# B&R Automation Studio project CleanChemi_SiteManagementSystem (part 12)

#### Status.st
```iecst
ACTION Modbus_Status_action:

	ModbusTcpMaster_HR[IdxSkids_HR]();

	//Reset Modbus buffer on connection timeout
	IF ModbusTcpMaster_HR[IdxSkids_HR].status = 50211 THEN
		brsmemset(ADR(gModbus_LR[IdxSkids_HR]),0,SIZEOF(gModbus_LR[IdxSkids_HR]));
	END_IF;

	// --------------------------------------------------------------------
	// Reset last error information
	// --------------------------------------------------------------------
	IF(reset_error) THEN
		brsmemset(ADR(ModbusTcpMaster_HR[IdxSkids_HR].last_error), 0, 2);
		reset_error := 0;
	END_IF

	// --------------------------------------------------------------------
	// Final Variable Mapping AND Data Conversion - READ
	// --------------------------------------------------------------------

	// AS Block 1 - 6000 DOSING INT
	gSkid_HR[IdxSkids_HR].Pmax_General_Variables.UNIT_ID := gModbus_HR[IdxSkids_HR].Modbus_PeroxyMAX.Block1_Int[0];
	gSkid_HR[IdxSkids_HR].Pmax_General_Variables.USER_ID := gModbus_HR[IdxSkids_HR].Modbus_PeroxyMAX.Block1_Int[2];
	gSkid_HR[IdxSkids_HR].Pmax_General_Variables.USER_ACCESS := gModbus_HR[IdxSkids_HR].Modbus_PeroxyMAX.Block1_Int[4];
	gSkid_HR[IdxSkids_HR].Pmax_General_Variables.PMAX_HOA := gModbus_HR[IdxSkids_HR].Modbus_PeroxyMAX.Block1_Int[6];
	gSkid_HR[IdxSkids_HR].Pmax_General_Variables.PMAX_STATUS := gModbus_HR[IdxSkids_HR].Modbus_PeroxyMAX.Block1_Int[8];
	gSkid_HR[IdxSkids_HR].Pmax_General_Variables.SCREEN_LOCK := INT_TO_BOOL(gModbus_HR[IdxSkids_HR].Modbus_PeroxyMAX.Block1_Int[10]);
	gSkid_HR[IdxSkids_HR].Pmax_General_Variables.HEARTBEAT := gModbus_HR[IdxSkids_HR].Modbus_PeroxyMAX.Block1_Int[12];

	gSkid_HR[IdxSkids_HR].Pmax_Pump_101.P101_XS := gModbus_HR[IdxSkids_HR].Modbus_PeroxyMAX.Block1_Int[20];
	gSkid_HR[IdxSkids_HR].Sensor_Variables.XV101 := gModbus_HR[IdxSkids_HR].Modbus_PeroxyMAX.Block1_Int[22];
	gSkid_HR[IdxSkids_HR].Sensor_Variables.XV101_ENABLE := gModbus_HR[IdxSkids_HR].Modbus_PeroxyMAX.Block1_Int[24];
	gSkid_HR[IdxSkids_HR].Pmax_Pump_101.P101_AUTOCAL := gModbus_HR[IdxSkids_HR].Modbus_PeroxyMAX.Block1_Int[26];

	gSkid_HR[IdxSkids_HR].Pmax_Pump_102.P102_XS := gModbus_HR[IdxSkids_HR].Modbus_PeroxyMAX.Block1_Int[32];
	gSkid_HR[IdxSkids_HR].Pmax_Pump_102.P102_WARN := gModbus_HR[IdxSkids_HR].Modbus_PeroxyMAX.Block1_Int[34];
	gSkid_HR[IdxSkids_HR].Pmax_Pump_102.P102_ALARM := gModbus_HR[IdxSkids_HR].Modbus_PeroxyMAX.Block1_Int[36];
	gSkid_HR[IdxSkids_HR].Sensor_Variables.XV102 := gModbus_HR[IdxSkids_HR].Modbus_PeroxyMAX.Block1_Int[38];
	gSkid_HR[IdxSkids_HR].Pmax_Pump_102.P102_AUTOCAL := gModbus_HR[IdxSkids_HR].Modbus_PeroxyMAX.Block1_Int[40];

	gSkid_HR[IdxSkids_HR].Pmax_Pump_103.P103_XS := gModbus_HR[IdxSkids_HR].Modbus_PeroxyMAX.Block1_Int[48];
	gSkid_HR[IdxSkids_HR].Pmax_Pump_103.P103_WARN := gModbus_HR[IdxSkids_HR].Modbus_PeroxyMAX.Block1_Int[50];
	gSkid_HR[IdxSkids_HR].Pmax_Pump_103.P103_ALARM := gModbus_HR[IdxSkids_HR].Modbus_PeroxyMAX.Block1_Int[52];
	gSkid_HR[IdxSkids_HR].Sensor_Variables.XV103 := gModbus_HR[IdxSkids_HR].Modbus_PeroxyMAX.Block1_Int[54];
	gSkid_HR[IdxSkids_HR].Pmax_Pump_103.P103_AUTOCAL := gModbus_HR[IdxSkids_HR].Modbus_PeroxyMAX.Block1_Int[56];

	gSkid_HR[IdxSkids_HR].Pmax_Pump_104.P104_XS := gModbus_HR[IdxSkids_HR].Modbus_PeroxyMAX.Block1_Int[64];
	gSkid_HR[IdxSkids_HR].Pmax_Pump_104.P104_WARN := gModbus_HR[IdxSkids_HR].Modbus_PeroxyMAX.Block1_Int[66];
	gSkid_HR[IdxSkids_HR].Pmax_Pump_104.P104_ALARM := gModbus_HR[IdxSkids_HR].Modbus_PeroxyMAX.Block1_Int[68];
	gSkid_HR[IdxSkids_HR].Sensor_Variables.XV104 := gModbus_HR[IdxSkids_HR].Modbus_PeroxyMAX.Block1_Int[70];
	gSkid_HR[IdxSkids_HR].Pmax_Pump_104.P104_AUTOCAL := gModbus_HR[IdxSkids_HR].Modbus_PeroxyMAX.Block1_Int[72];
	gSkid_HR[IdxSkids_HR].Pmax_Pump_104.P104_AUTOCAL_PV := gModbus_HR[IdxSkids_HR].Modbus_PeroxyMAX.Block1_Int[74];

	// AS Block 2 - 6000 DOSING INT - SPARE
	//:= gModbus_HR[IdxSkids_HR].Modbus_PeroxyMAX.Block2_Int[0];

	// AS Block 3 - 6000 DOSING REAL
	gSkid_HR[IdxSkids_HR].ConversionRatios.EFF_1:= IDEC_REAL_Conv(gModbus_HR[IdxSkids_HR].Modbus_PeroxyMAX.Block3_Real[0]);
	gSkid_HR[IdxSkids_HR].ConversionRatios.EFF_2:= IDEC_REAL_Conv(gModbus_HR[IdxSkids_HR].Modbus_PeroxyMAX.Block3_Real[1]);
	gSkid_HR[IdxSkids_HR].ConversionRatios.NAOH_TO_H2O2:= IDEC_REAL_Conv(gModbus_HR[IdxSkids_HR].Modbus_PeroxyMAX.Block3_Real[2]);
	gSkid_HR[IdxSkids_HR].ConversionRatios.TRI_TO_H2O2:= IDEC_REAL_Conv(gModbus_HR[IdxSkids_HR].Modbus_PeroxyMAX.Block3_Real[3]);
	gSkid_HR[IdxSkids_HR].ConversionRatios.NAOH_TO_TRI:= IDEC_REAL_Conv(gModbus_HR[IdxSkids_HR].Modbus_PeroxyMAX.Block3_Real[4]);

	gSkid_HR[IdxSkids_HR].Pmax_General_Variables.PMAX_CONC:= IDEC_REAL_Conv(gModbus_HR[IdxSkids_HR].Modbus_PeroxyMAX.Block3_Real[8]);
	gSkid_HR[IdxSkids_HR].Pmax_General_Variables.PMAX_RATE:= IDEC_REAL_Conv(gModbus_HR[IdxSkids_HR].Modbus_PeroxyMAX.Block3_Real[9]);
	gSkid_HR[IdxSkids_HR].Pmax_General_Variables.PMAX_PV:= IDEC_REAL_Conv(gModbus_HR[IdxSkids_HR].Modbus_PeroxyMAX.Block3_Real[10]);
	gSkid_HR[IdxSkids_HR].Pmax_General_Variables.NAOH_CONC:= IDEC_REAL_Conv(gModbus_HR[IdxSkids_HR].Modbus_PeroxyMAX.Block3_Real[11]);
	gSkid_HR[IdxSkids_HR].Pmax_General_Variables.NAOH_CONC_OD:= IDEC_REAL_Conv(gModbus_HR[IdxSkids_HR].Modbus_PeroxyMAX.Block3_Real[12]);
	gSkid_HR[IdxSkids_HR].Pmax_General_Variables.HP_CONC:= IDEC_REAL_Conv(gModbus_HR[IdxSkids_HR].Modbus_PeroxyMAX.Block3_Real[13]);
	gSkid_HR[IdxSkids_HR].Pmax_General_Variables.HP_CONC_OD:= IDEC_REAL_Conv(gModbus_HR[IdxSkids_HR].Modbus_PeroxyMAX.Block3_Real[14]);

	gSkid_HR[IdxSkids_HR].Pmax_Pump_101.P101_SP:= IDEC_REAL_Conv(gModbus_HR[IdxSkids_HR].Modbus_PeroxyMAX.Block3_Real[21]);
	gSkid_HR[IdxSkids_HR].Pmax_Pump_101.P101_PV:= IDEC_REAL_Conv(gModbus_HR[IdxSkids_HR].Modbus_PeroxyMAX.Block3_Real[22]);
	gSkid_HR[IdxSkids_HR].Pmax_Pump_101.P101_OP:= IDEC_REAL_Conv(gModbus_HR[IdxSkids_HR].Modbus_PeroxyMAX.Block3_Real[23]);
	gSkid_HR[IdxSkids_HR].Pmax_Pump_101.P101_FQ:= IDEC_REAL_Conv(gModbus_HR[IdxSkids_HR].Modbus_PeroxyMAX.Block3_Real[24]);
	gSkid_HR[IdxSkids_HR].Pmax_Pump_101.P101_TI:= IDEC_REAL_Conv(gModbus_HR[IdxSkids_HR].Modbus_PeroxyMAX.Block3_Real[25]);
	gSkid_HR[IdxSkids_HR].Pmax_Pump_101.P101_PI:= IDEC_REAL_Conv(gModbus_HR[IdxSkids_HR].Modbus_PeroxyMAX.Block3_Real[26]);
	gSkid_HR[IdxSkids_HR].Pmax_Pump_101.P101_PFI:= IDEC_REAL_Conv(gModbus_HR[IdxSkids_HR].Modbus_PeroxyMAX.Block3_Real[27]);
	gSkid_HR[IdxSkids_HR].Pmax_Pump_101.P101_LS:= IDEC_REAL_Conv(gModbus_HR[IdxSkids_HR].Modbus_PeroxyMAX.Block3_Real[28]);
	gSkid_HR[IdxSkids_HR].Pmax_Pump_101.P101_GAIN:= IDEC_REAL_Conv(gModbus_HR[IdxSkids_HR].Modbus_PeroxyMAX.Block3_Real[29]);
	gSkid_HR[IdxSkids_HR].Pmax_Pump_101.P101_STEPADJ:= IDEC_REAL_Conv(gModbus_HR[IdxSkids_HR].Modbus_PeroxyMAX.Block3_Real[30]);
	gSkid_HR[IdxSkids_HR].Pmax_Pump_101.P101_TOTALADJ:= IDEC_REAL_Conv(gModbus_HR[IdxSkids_HR].Modbus_PeroxyMAX.Block3_Real[31]);

	gSkid_HR[IdxSkids_HR].Pmax_Pump_101B.P101B_OP:= IDEC_REAL_Conv(gModbus_HR[IdxSkids_HR].Modbus_PeroxyMAX.Block3_Real[35]);
	gSkid_HR[IdxSkids_HR].Pmax_Pump_101B.P101B_PFI:= IDEC_REAL_Conv(gModbus_HR[IdxSkids_HR].Modbus_PeroxyMAX.Block3_Real[36]);
	gSkid_HR[IdxSkids_HR].Pmax_Pump_101B.P101B_SP:= IDEC_REAL_Conv(gModbus_HR[IdxSkids_HR].Modbus_PeroxyMAX.Block3_Real[37]);
	gSkid_HR[IdxSkids_HR].Pmax_Pump_101B.P101B_LS:= IDEC_REAL_Conv(gModbus_HR[IdxSkids_HR].Modbus_PeroxyMAX.Block3_Real[38]);

	gSkid_HR[IdxSkids_HR].Pmax_Pump_102.P102_SP:= IDEC_REAL_Conv(gModbus_HR[IdxSkids_HR].Modbus_PeroxyMAX.Block3_Real[45]);
	gSkid_HR[IdxSkids_HR].Pmax_Pump_102.P102_PV:= IDEC_REAL_Conv(gModbus_HR[IdxSkids_HR].Modbus_PeroxyMAX.Block3_Real[46]);
	gSkid_HR[IdxSkids_HR].Pmax_Pump_102.P102_OP:= IDEC_REAL_Conv(gModbus_HR[IdxSkids_HR].Modbus_PeroxyMAX.Block3_Real[47]);
	gSkid_HR[IdxSkids_HR].Pmax_Pump_102.P102_PFI:= IDEC_REAL_Conv(gModbus_HR[IdxSkids_HR].Modbus_PeroxyMAX.Block3_Real[48]);
	gSkid_HR[IdxSkids_HR].Pmax_Pump_102.P102_FQ:= IDEC_REAL_Conv(gModbus_HR[IdxSkids_HR].Modbus_PeroxyMAX.Block3_Real[49]);
	gSkid_HR[IdxSkids_HR].Pmax_Pump_102.P102_PFQ:= IDEC_REAL_Conv(gModbus_HR[IdxSkids_HR].Modbus_PeroxyMAX.Block3_Real[50]);
	gSkid_HR[IdxSkids_HR].Pmax_Pump_102.P102_PPI:= IDEC_REAL_Conv(gModbus_HR[IdxSkids_HR].Modbus_PeroxyMAX.Block3_Real[51]);
	gSkid_HR[IdxSkids_HR].Pmax_Pump_102.P102_TI:= IDEC_REAL_Conv(gModbus_HR[IdxSkids_HR].Modbus_PeroxyMAX.Block3_Real[52]);
	gSkid_HR[IdxSkids_HR].Pmax_Pump_102.P102_PI:= IDEC_REAL_Conv(gModbus_HR[IdxSkids_HR].Modbus_PeroxyMAX.Block3_Real[53]);
	gSkid_HR[IdxSkids_HR].Pmax_Pump_102.P102_LS:= IDEC_REAL_Conv(gModbus_HR[IdxSkids_HR].Modbus_PeroxyMAX.Block3_Real[54]);
	gSkid_HR[IdxSkids_HR].Pmax_Pump_102.P102_GAIN:= IDEC_REAL_Conv(gModbus_HR[IdxSkids_HR].Modbus_PeroxyMAX.Block3_Real[55]);
	gSkid_HR[IdxSkids_HR].Pmax_Pump_102.P102_STEPADJ:= IDEC_REAL_Conv(gModbus_HR[IdxSkids_HR].Modbus_PeroxyMAX.Block3_Real[56]);
	gSkid_HR[IdxSkids_HR].Pmax_Pump_102.P102_TOTALADJ:= IDEC_REAL_Conv(gModbus_HR[IdxSkids_HR].Modbus_PeroxyMAX.Block3_Real[57]);

	gSkid_HR[IdxSkids_HR].Pmax_Pump_103.P103_SP:= IDEC_REAL_Conv(gModbus_HR[IdxSkids_HR].Modbus_PeroxyMAX.Block3_Real[59]);
	gSkid_HR[IdxSkids_HR].Pmax_Pump_103.P103_PV:= IDEC_REAL_Conv(gModbus_HR[IdxSkids_HR].Modbus_PeroxyMAX.Block3_Real[60]);
	gSkid_HR[IdxSkids_HR].Pmax_Pump_103.P103_OP:= IDEC_REAL_Conv(gModbus_HR[IdxSkids_HR].Modbus_PeroxyMAX.Block3_Real[61]);
	gSkid_HR[IdxSkids_HR].Pmax_Pump_103.P103_PFI:= IDEC_REAL_Conv(gModbus_HR[IdxSkids_HR].Modbus_PeroxyMAX.Block3_Real[62]);

	// AS Block 4 - 6000 DOSING REAL
	gSkid_HR[IdxSkids_HR].Pmax_Pump_103.P103_FQ:= IDEC_REAL_Conv(gModbus_HR[IdxSkids_HR].Modbus_PeroxyMAX.Block4_Real[0]);
	gSkid_HR[IdxSkids_HR].Pmax_Pump_103.P103_PFQ:= IDEC_REAL_Conv(gModbus_HR[IdxSkids_HR].Modbus_PeroxyMAX.Block4_Real[1]);
	gSkid_HR[IdxSkids_HR].Pmax_Pump_103.P103_PPI:= IDEC_REAL_Conv(gModbus_HR[IdxSkids_HR].Modbus_PeroxyMAX.Block4_Real[2]);
	gSkid_HR[IdxSkids_HR].Pmax_Pump_103.P103_TI:= IDEC_REAL_Conv(gModbus_HR[IdxSkids_HR].Modbus_PeroxyMAX.Block4_Real[3]);
	gSkid_HR[IdxSkids_HR].Pmax_Pump_103.P103_PI:= IDEC_REAL_Conv(gModbus_HR[IdxSkids_HR].Modbus_PeroxyMAX.Block4_Real[4]);
	gSkid_HR[IdxSkids_HR].Pmax_Pump_103.P103_LS:= IDEC_REAL_Conv(gModbus_HR[IdxSkids_HR].Modbus_PeroxyMAX.Block4_Real[5]);
	gSkid_HR[IdxSkids_HR].Pmax_Pump_103.P103_GAIN:= IDEC_REAL_Conv(gModbus_HR[IdxSkids_HR].Modbus_PeroxyMAX.Block3_Real[6]);
	gSkid_HR[IdxSkids_HR].Pmax_Pump_103.P103_STEPADJ:= IDEC_REAL_Conv(gModbus_HR[IdxSkids_HR].Modbus_PeroxyMAX.Block3_Real[7]);
	gSkid_HR[IdxSkids_HR].Pmax_Pump_103.P103_TOTALADJ:= IDEC_REAL_Conv(gModbus_HR[IdxSkids_HR].Modbus_PeroxyMAX.Block3_Real[8]);

	gSkid_HR[IdxSkids_HR].Pmax_Pump_104.P104_SP:= IDEC_REAL_Conv(gModbus_HR[IdxSkids_HR].Modbus_PeroxyMAX.Block4_Real[10]);
	gSkid_HR[IdxSkids_HR].Pmax_Pump_104.P104_PV:= IDEC_REAL_Conv(gModbus_HR[IdxSkids_HR].Modbus_PeroxyMAX.Block4_Real[11]);
	gSkid_HR[IdxSkids_HR].Pmax_Pump_104.P104_OP:= IDEC_REAL_Conv(gModbus_HR[IdxSkids_HR].Modbus_PeroxyMAX.Block4_Real[12]);
	gSkid_HR[IdxSkids_HR].Pmax_Pump_104.P104_PFI:= IDEC_REAL_Conv(gModbus_HR[IdxSkids_HR].Modbus_PeroxyMAX.Block4_Real[13]);
	gSkid_HR[IdxSkids_HR].Pmax_Pump_104.P104_FQ:= IDEC_REAL_Conv(gModbus_HR[IdxSkids_HR].Modbus_PeroxyMAX.Block4_Real[14]);
	gSkid_HR[IdxSkids_HR].Pmax_Pump_104.P104_PFQ:= IDEC_REAL_Conv(gModbus_HR[IdxSkids_HR].Modbus_PeroxyMAX.Block4_Real[15]);
	gSkid_HR[IdxSkids_HR].Pmax_Pump_104.P104_PPI:= IDEC_REAL_Conv(gModbus_HR[IdxSkids_HR].Modbus_PeroxyMAX.Block4_Real[16]);
	gSkid_HR[IdxSkids_HR].Pmax_Pump_104.P104_PI:= IDEC_REAL_Conv(gModbus_HR[IdxSkids_HR].Modbus_PeroxyMAX.Block4_Real[17]);
	gSkid_HR[IdxSkids_HR].Pmax_Pump_104.P104_LS:= IDEC_REAL_Conv(gModbus_HR[IdxSkids_HR].Modbus_PeroxyMAX.Block4_Real[18]);
	gSkid_HR[IdxSkids_HR].Pmax_Pump_104.P104_GAIN:= IDEC_REAL_Conv(gModbus_HR[IdxSkids_HR].Modbus_PeroxyMAX.Block3_Real[19]);
	gSkid_HR[IdxSkids_HR].Pmax_Pump_104.P104_STEPADJ:= IDEC_REAL_Conv(gModbus_HR[IdxSkids_HR].Modbus_PeroxyMAX.Block3_Real[20]);
	gSkid_HR[IdxSkids_HR].Pmax_Pump_104.P104_TOTALADJ:= IDEC_REAL_Conv(gModbus_HR[IdxSkids_HR].Modbus_PeroxyMAX.Block3_Real[21]);

	gSkid_HR[IdxSkids_HR].Sensor_Variables.CD101:= IDEC_REAL_Conv(gModbus_HR[IdxSkids_HR].Modbus_PeroxyMAX.Block4_Real[24]);
	gSkid_HR[IdxSkids_HR].Sensor_Variables.CD101_SP:= IDEC_REAL_Conv(gModbus_HR[IdxSkids_HR].Modbus_PeroxyMAX.Block4_Real[25]);
	gSkid_HR[IdxSkids_HR].Sensor_Variables.CD102:= IDEC_REAL_Conv(gModbus_HR[IdxSkids_HR].Modbus_PeroxyMAX.Block4_Real[26]);
	gSkid_HR[IdxSkids_HR].Sensor_Variables.CD102_SP:= IDEC_REAL_Conv(gModbus_HR[IdxSkids_HR].Modbus_PeroxyMAX.Block4_Real[27]);
	gSkid_HR[IdxSkids_HR].Sensor_Variables.CD103:= IDEC_REAL_Conv(gModbus_HR[IdxSkids_HR].Modbus_PeroxyMAX.Block4_Real[28]);
	gSkid_HR[IdxSkids_HR].Sensor_Variables.CD103_SP:= IDEC_REAL_Conv(gModbus_HR[IdxSkids_HR].Modbus_PeroxyMAX.Block4_Real[29]);

	gSkid_HR[IdxSkids_HR].Sensor_Variables.CD101_TI:= IDEC_REAL_Conv(gModbus_HR[IdxSkids_HR].Modbus_PeroxyMAX.Block4_Real[36]);
	gSkid_HR[IdxSkids_HR].Sensor_Variables.CD102_TI:= IDEC_REAL_Conv(gModbus_HR[IdxSkids_HR].Modbus_PeroxyMAX.Block4_Real[37]);
	gSkid_HR[IdxSkids_HR].Sensor_Variables.CD103_TI:= IDEC_REAL_Conv(gModbus_HR[IdxSkids_HR].Modbus_PeroxyMAX.Block4_Real[38]);

	gSkid_HR[IdxSkids_HR].Pmax_General_Variables.HMI_REV_A:= IDEC_REAL_Conv(gModbus_HR[IdxSkids_HR].Modbus_PeroxyMAX.Block4_Real[45]);
	gSkid_HR[IdxSkids_HR].Pmax_General_Variables.HMI_REV_B:= IDEC_REAL_Conv(gModbus_HR[IdxSkids_HR].Modbus_PeroxyMAX.Block4_Real[46]);
	gSkid_HR[IdxSkids_HR].Pmax_General_Variables.PLC_REV_A:= IDEC_REAL_Conv(gModbus_HR[IdxSkids_HR].Modbus_PeroxyMAX.Block4_Real[47]);
	gSkid_HR[IdxSkids_HR].Pmax_General_Variables.PLC_REV_B:= IDEC_REAL_Conv(gModbus_HR[IdxSkids_HR].Modbus_PeroxyMAX.Block4_Real[48]);

	gSkid_HR[IdxSkids_HR].BufferTank.BT_PERCENT:= IDEC_REAL_Conv(gModbus_HR[IdxSkids_HR].Modbus_PeroxyMAX.Block4_Real[50]);
	gSkid_HR[IdxSkids_HR].BufferTank.LI200:= IDEC_REAL_Conv(gModbus_HR[IdxSkids_HR].Modbus_PeroxyMAX.Block4_Real[51]);
	gSkid_HR[IdxSkids_HR].BufferTank.LSHH200:= IDEC_REAL_Conv(gModbus_HR[IdxSkids_HR].Modbus_PeroxyMAX.Block4_Real[52]);
	gSkid_HR[IdxSkids_HR].BufferTank.DRAINTIME_SP:= IDEC_REAL_Conv(gModbus_HR[IdxSkids_HR].Modbus_PeroxyMAX.Block4_Real[53]);
	gSkid_HR[IdxSkids_HR].BufferTank.DRAINTIME_PV:= IDEC_REAL_Conv(gModbus_HR[IdxSkids_HR].Modbus_PeroxyMAX.Block4_Real[54]);
	gSkid_HR[IdxSkids_HR].BufferTank.FILLTIME_SP:= IDEC_REAL_Conv(gModbus_HR[IdxSkids_HR].Modbus_PeroxyMAX.Block4_Real[55]);
	gSkid_HR[IdxSkids_HR].BufferTank.FILLTIME_PV:= IDEC_REAL_Conv(gModbus_HR[IdxSkids_HR].Modbus_PeroxyMAX.Block4_Real[56]);

	// AS Block 5 - 6000 DOSING REAL - SPARE
	//:= IDEC_REAL_Conv(gModbus_HR[IdxSkids_HR].Modbus_PeroxyMAX.Block5_Real[0]);

	// AS Block 6 - 7000 DOSING INT
	gSkid_HR[IdxSkids_HR].Pmax_General_Variables.UNIT_ID_DOSE := gModbus_HR[IdxSkids_HR].Modbus_Dosing.Block6_Int[0];

	gSkid_HR[IdxSkids_HR].Dosing_Pump_201.P201_XS := gModbus_HR[IdxSkids_HR].Modbus_Dosing.Block6_Int[6];
	gSkid_HR[IdxSkids_HR].Dosing_Pump_201.P201_HOA := gModbus_HR[IdxSkids_HR].Modbus_Dosing.Block6_Int[8];
	gSkid_HR[IdxSkids_HR].Dosing_Pump_201.P201_CHEM := gModbus_HR[IdxSkids_HR].Modbus_Dosing.Block6_Int[10];
	gSkid_HR[IdxSkids_HR].Dosing_Pump_201.P201_ENABLE := gModbus_HR[IdxSkids_HR].Modbus_Dosing.Block6_Int[12];
	gSkid_HR[IdxSkids_HR].Dosing_Pump_201.P201_ADJ := gModbus_HR[IdxSkids_HR].Modbus_Dosing.Block6_Int[14];
	gSkid_HR[IdxSkids_HR].Dosing_Pump_201.P201_PTYPE := gModbus_HR[IdxSkids_HR].Modbus_Dosing.Block6_Int[16];
	gSkid_HR[IdxSkids_HR].Dosing_Pump_201.P201_WARN := gModbus_HR[IdxSkids_HR].Modbus_Dosing.Block6_Int[18];
	gSkid_HR[IdxSkids_HR].Dosing_Pump_201.P201_ALARM := gModbus_HR[IdxSkids_HR].Modbus_Dosing.Block6_Int[20];
	gSkid_HR[IdxSkids_HR].Sensor_Variables.XV201 := gModbus_HR[IdxSkids_HR].Modbus_Dosing.Block6_Int[22];
	gSkid_HR[IdxSkids_HR].Dosing_Pump_201.P201_AUTOCAL := gModbus_HR[IdxSkids_HR].Modbus_Dosing.Block6_Int[24];
	gSkid_HR[IdxSkids_HR].Dosing_Pump_201.P201_AUTOCAL_PV := gModbus_HR[IdxSkids_HR].Modbus_Dosing.Block6_Int[26];

	gSkid_HR[IdxSkids_HR].Dosing_Pump_202.P202_XS := gModbus_HR[IdxSkids_HR].Modbus_Dosing.Block6_Int[32];
	gSkid_HR[IdxSkids_HR].Dosing_Pump_202.P202_HOA := gModbus_HR[IdxSkids_HR].Modbus_Dosing.Block6_Int[34];
	gSkid_HR[IdxSkids_HR].Dosing_Pump_202.P202_CHEM := gModbus_HR[IdxSkids_HR].Modbus_Dosing.Block6_Int[36];
	gSkid_HR[IdxSkids_HR].Dosing_Pump_202.P202_ENABLE := gModbus_HR[IdxSkids_HR].Modbus_Dosing.Block6_Int[38];
	gSkid_HR[IdxSkids_HR].Dosing_Pump_202.P202_ADJ := gModbus_HR[IdxSkids_HR].Modbus_Dosing.Block6_Int[40];
	gSkid_HR[IdxSkids_HR].Dosing_Pump_202.P202_WARN := gModbus_HR[IdxSkids_HR].Modbus_Dosing.Block6_Int[42];
	gSkid_HR[IdxSkids_HR].Dosing_Pump_202.P202_ALARM := gModbus_HR[IdxSkids_HR].Modbus_Dosing.Block6_Int[44];
	gSkid_HR[IdxSkids_HR].Sensor_Variables.XV202 := gModbus_HR[IdxSkids_HR].Modbus_Dosing.Block6_Int[46];
	gSkid_HR[IdxSkids_HR].Dosing_Pump_202.P202_AUTOCAL := gModbus_HR[IdxSkids_HR].Modbus_Dosing.Block6_Int[48];
	gSkid_HR[IdxSkids_HR].Dosing_Pump_202.P202_AUTOCAL_PV := gModbus_HR[IdxSkids_HR].Modbus_Dosing.Block6_Int[50];

	gSkid_HR[IdxSkids_HR].Dosing_Pump_203.P203_XS := gModbus_HR[IdxSkids_HR].Modbus_Dosing.Block6_Int[56];
	gSkid_HR[IdxSkids_HR].Dosing_Pump_203.P203_HOA := gModbus_HR[IdxSkids_HR].Modbus_Dosing.Block6_Int[58];
	gSkid_HR[IdxSkids_HR].Dosing_Pump_203.P203_CHEM := gModbus_HR[IdxSkids_HR].Modbus_Dosing.Block6_Int[60];
	gSkid_HR[IdxSkids_HR].Dosing_Pump_203.P203_ENABLE := gModbus_HR[IdxSkids_HR].Modbus_Dosing.Block6_Int[62];
	gSkid_HR[IdxSkids_HR].Dosing_Pump_203.P203_ADJ := gModbus_HR[IdxSkids_HR].Modbus_Dosing.Block6_Int[64];
	gSkid_HR[IdxSkids_HR].Dosing_Pump_203.P203_WARN := gModbus_HR[IdxSkids_HR].Modbus_Dosing.Block6_Int[66];
	gSkid_HR[IdxSkids_HR].Dosing_Pump_203.P203_ALARM := gModbus_HR[IdxSkids_HR].Modbus_Dosing.Block6_Int[68];
	gSkid_HR[IdxSkids_HR].Sensor_Variables.XV203 := gModbus_HR[IdxSkids_HR].Modbus_Dosing.Block6_Int[70];
	gSkid_HR[IdxSkids_HR].Dosing_Pump_203.P203_AUTOCAL := gModbus_HR[IdxSkids_HR].Modbus_Dosing.Block6_Int[72];
	gSkid_HR[IdxSkids_HR].Dosing_Pump_203.P203_AUTOCAL_PV := gModbus_HR[IdxSkids_HR].Modbus_Dosing.Block6_Int[74];

	gSkid_HR[IdxSkids_HR].Dosing_Pump_204.P204_XS := gModbus_HR[IdxSkids_HR].Modbus_Dosing.Block6_Int[80];
	gSkid_HR[IdxSkids_HR].Dosing_Pump_204.P204_HOA := gModbus_HR[IdxSkids_HR].Modbus_Dosing.Block6_Int[82];
	gSkid_HR[IdxSkids_HR].Dosing_Pump_204.P204_CHEM := gModbus_HR[IdxSkids_HR].Modbus_Dosing.Block6_Int[84];
	gSkid_HR[IdxSkids_HR].Dosing_Pump_204.P204_ENABLE := gModbus_HR[IdxSkids_HR].Modbus_Dosing.Block6_Int[86];
	gSkid_HR[IdxSkids_HR].Dosing_Pump_204.P204_ADJ := gModbus_HR[IdxSkids_HR].Modbus_Dosing.Block6_Int[88];
	gSkid_HR[IdxSkids_HR].Dosing_Pump_204.P204_WARN := gModbus_HR[IdxSkids_HR].Modbus_Dosing.Block6_Int[90];
	gSkid_HR[IdxSkids_HR].Dosing_Pump_204.P204_ALARM := gModbus_HR[IdxSkids_HR].Modbus_Dosing.Block6_Int[92];
	gSkid_HR[IdxSkids_HR].Sensor_Variables.XV204 := gModbus_HR[IdxSkids_HR].Modbus_Dosing.Block6_Int[94];
	gSkid_HR[IdxSkids_HR].Dosing_Pump_204.P204_AUTOCAL := gModbus_HR[IdxSkids_HR].Modbus_Dosing.Block6_Int[96];
	gSkid_HR[IdxSkids_HR].Dosing_Pump_204.P204_AUTOCAL_PV := gModbus_HR[IdxSkids_HR].Modbus_Dosing.Block6_Int[98];

	gSkid_HR[IdxSkids_HR].Dosing_Pump_205.P205_XS := gModbus_HR[IdxSkids_HR].Modbus_Dosing.Block6_Int[104];
	gSkid_HR[IdxSkids_HR].Dosing_Pump_205.P205_HOA := gModbus_HR[IdxSkids_HR].Modbus_Dosing.Block6_Int[106];
	gSkid_HR[IdxSkids_HR].Dosing_Pump_205.P205_CHEM := gModbus_HR[IdxSkids_HR].Modbus_Dosing.Block6_Int[108];

	// AS Block 7 - 7000 DOSING INT
	gSkid_HR[IdxSkids_HR].Dosing_Pump_206.P206_XS := gModbus_HR[IdxSkids_HR].Modbus_Dosing.Block7_Int[2];
	gSkid_HR[IdxSkids_HR].Dosing_Pump_206.P206_HOA := gModbus_HR[IdxSkids_HR].Modbus_Dosing.Block7_Int[4];
	gSkid_HR[IdxSkids_HR].Dosing_Pump_206.P206_CHEM := gModbus_HR[IdxSkids_HR].Modbus_Dosing.Block7_Int[6];

	gSkid_HR[IdxSkids_HR].Dosing_Pump_207.P207_XS := gModbus_HR[IdxSkids_HR].Modbus_Dosing.Block7_Int[26];
	gSkid_HR[IdxSkids_HR].Dosing_Pump_207.P207_HOA := gModbus_HR[IdxSkids_HR].Modbus_Dosing.Block7_Int[28];
	gSkid_HR[IdxSkids_HR].Dosing_Pump_207.P207_CHEM := gModbus_HR[IdxSkids_HR].Modbus_Dosing.Block7_Int[30];

	gSkid_HR[IdxSkids_HR].Dosing_Pump_208.P208_XS := gModbus_HR[IdxSkids_HR].Modbus_Dosing.Block7_Int[50];
	gSkid_HR[IdxSkids_HR].Dosing_Pump_208.P208_HOA := gModbus_HR[IdxSkids_HR].Modbus_Dosing.Block7_Int[52];
	gSkid_HR[IdxSkids_HR].Dosing_Pump_208.P208_CHEM := gModbus_HR[IdxSkids_HR].Modbus_Dosing.Block7_Int[54];

	gSkid_HR[IdxSkids_HR].Sensor_Variables.SERNSORS_CONFIG := gModbus_HR[IdxSkids_HR].Modbus_Dosing.Block7_Int[104];

	gSkid_HR[IdxSkids_HR].Sensor_Variables.FI301_MODE := gModbus_HR[IdxSkids_HR].Modbus_Dosing.Block7_Int[118];
	gSkid_HR[IdxSkids_HR].Sensor_Variables.FI302_MODE := gModbus_HR[IdxSkids_HR].Modbus_Dosing.Block7_Int[120];
	gSkid_HR[IdxSkids_HR].Sensor_Variables.FI303_MODE := gModbus_HR[IdxSkids_HR].Modbus_Dosing.Block7_Int[122];
	gSkid_HR[IdxSkids_HR].Sensor_Variables.FI304_MODE := gModbus_HR[IdxSkids_HR].Modbus_Dosing.Block7_Int[124];

	// AS Block 8 - 7000 DOSING REAL
	gSkid_HR[IdxSkids_HR].Dosing_Pump_201.P201_REF_SENSOR := IDEC_REAL_Conv(gModbus_HR[IdxSkids_HR].Modbus_Dosing.Block8_Real[0]);
	gSkid_HR[IdxSkids_HR].Dosing_Pump_201.P201_CONC := IDEC_REAL_Conv(gModbus_HR[IdxSkids_HR].Modbus_Dosing.Block8_Real[1]);
	gSkid_HR[IdxSkids_HR].Dosing_Pump_201.P201_PPM := IDEC_REAL_Conv(gModbus_HR[IdxSkids_HR].Modbus_Dosing.Block8_Real[2]);
	gSkid_HR[IdxSkids_HR].Dosing_Pump_201.P201_APPM := IDEC_REAL_Conv(gModbus_HR[IdxSkids_HR].Modbus_Dosing.Block8_Real[3]);
	gSkid_HR[IdxSkids_HR].Dosing_Pump_201.P201_SP := IDEC_REAL_Conv(gModbus_HR[IdxSkids_HR].Modbus_Dosing.Block8_Real[4]);
	gSkid_HR[IdxSkids_HR].Dosing_Pump_201.P201_PV := IDEC_REAL_Conv(gModbus_HR[IdxSkids_HR].Modbus_Dosing.Block8_Real[5]);
	gSkid_HR[IdxSkids_HR].Dosing_Pump_201.P201_OP := IDEC_REAL_Conv(gModbus_HR[IdxSkids_HR].Modbus_Dosing.Block8_Real[6]);
	gSkid_HR[IdxSkids_HR].Dosing_Pump_201.P201_PFI := IDEC_REAL_Conv(gModbus_HR[IdxSkids_HR].Modbus_Dosing.Block8_Real[7]);
	gSkid_HR[IdxSkids_HR].Dosing_Pump_201.P201_FQ := IDEC_REAL_Conv(gModbus_HR[IdxSkids_HR].Modbus_Dosing.Block8_Real[8]);
	gSkid_HR[IdxSkids_HR].Dosing_Pump_201.P201_PI := IDEC_REAL_Conv(gModbus_HR[IdxSkids_HR].Modbus_Dosing.Block8_Real[9]);
	gSkid_HR[IdxSkids_HR].Dosing_Pump_201.P201_TI := IDEC_REAL_Conv(gModbus_HR[IdxSkids_HR].Modbus_Dosing.Block8_Real[10]);
	gSkid_HR[IdxSkids_HR].Dosing_Pump_201.P201_PFQ := IDEC_REAL_Conv(gModbus_HR[IdxSkids_HR].Modbus_Dosing.Block8_Real[11]);
	gSkid_HR[IdxSkids_HR].Dosing_Pump_201.P201_PPI := IDEC_REAL_Conv(gModbus_HR[IdxSkids_HR].Modbus_Dosing.Block8_Real[12]);
	gSkid_HR[IdxSkids_HR].Dosing_Pump_201.P201_LS := IDEC_REAL_Conv(gModbus_HR[IdxSkids_HR].Modbus_Dosing.Block8_Real[13]);
	gSkid_HR[IdxSkids_HR].Dosing_Pump_201.P201_ASP := IDEC_REAL_Conv(gModbus_HR[IdxSkids_HR].Modbus_Dosing.Block8_Real[14]);
	gSkid_HR[IdxSkids_HR].Dosing_Pump_201.P201_GAIN := IDEC_REAL_Conv(gModbus_HR[IdxSkids_HR].Modbus_Dosing.Block8_Real[15]);
	gSkid_HR[IdxSkids_HR].Dosing_Pump_201.P201_STEPADJ := IDEC_REAL_Conv(gModbus_HR[IdxSkids_HR].Modbus_Dosing.Block8_Real[16]);
	gSkid_HR[IdxSkids_HR].Dosing_Pump_201.P201_TOTALADJ := IDEC_REAL_Conv(gModbus_HR[IdxSkids_HR].Modbus_Dosing.Block8_Real[17]);

	gSkid_HR[IdxSkids_HR].Dosing_Pump_202.P202_REF_SENSOR := IDEC_REAL_Conv(gModbus_HR[IdxSkids_HR].Modbus_Dosing.Block8_Real[19]);
	gSkid_HR[IdxSkids_HR].Dosing_Pump_202.P202_CONC := IDEC_REAL_Conv(gModbus_HR[IdxSkids_HR].Modbus_Dosing.Block8_Real[20]);
	gSkid_HR[IdxSkids_HR].Dosing_Pump_202.P202_PPM := IDEC_REAL_Conv(gModbus_HR[IdxSkids_HR].Modbus_Dosing.Block8_Real[21]);
	gSkid_HR[IdxSkids_HR].Dosing_Pump_202.P202_APPM := IDEC_REAL_Conv(gModbus_HR[IdxSkids_HR].Modbus_Dosing.Block8_Real[22]);
	gSkid_HR[IdxSkids_HR].Dosing_Pump_202.P202_SP := IDEC_REAL_Conv(gModbus_HR[IdxSkids_HR].Modbus_Dosing.Block8_Real[23]);
	gSkid_HR[IdxSkids_HR].Dosing_Pump_202.P202_PV := IDEC_REAL_Conv(gModbus_HR[IdxSkids_HR].Modbus_Dosing.Block8_Real[24]);
	gSkid_HR[IdxSkids_HR].Dosing_Pump_202.P202_OP := IDEC_REAL_Conv(gModbus_HR[IdxSkids_HR].Modbus_Dosing.Block8_Real[25]);
	gSkid_HR[IdxSkids_HR].Dosing_Pump_202.P202_PFI := IDEC_REAL_Conv(gModbus_HR[IdxSkids_HR].Modbus_Dosing.Block8_Real[26]);
	gSkid_HR[IdxSkids_HR].Dosing_Pump_202.P202_FQ := IDEC_REAL_Conv(gModbus_HR[IdxSkids_HR].Modbus_Dosing.Block8_Real[27]);
	gSkid_HR[IdxSkids_HR].Dosing_Pump_202.P202_PI := IDEC_REAL_Conv(gModbus_HR[IdxSkids_HR].Modbus_Dosing.Block8_Real[28]);
	gSkid_HR[IdxSkids_HR].Dosing_Pump_202.P202_TI := IDEC_REAL_Conv(gModbus_HR[IdxSkids_HR].Modbus_Dosing.Block8_Real[29]);
	gSkid_HR[IdxSkids_HR].Dosing_Pump_202.P202_PFQ := IDEC_REAL_Conv(gModbus_HR[IdxSkids_HR].Modbus_Dosing.Block8_Real[30]);
	gSkid_HR[IdxSkids_HR].Dosing_Pump_202.P202_PPI := IDEC_REAL_Conv(gModbus_HR[IdxSkids_HR].Modbus_Dosing.Block8_Real[31]);
	gSkid_HR[IdxSkids_HR].Dosing_Pump_202.P202_LS := IDEC_REAL_Conv(gModbus_HR[IdxSkids_HR].Modbus_Dosing.Block8_Real[32]);
	gSkid_HR[IdxSkids_HR].Dosing_Pump_202.P202_ASP := IDEC_REAL_Conv(gModbus_HR[IdxSkids_HR].Modbus_Dosing.Block8_Real[33]);
	gSkid_HR[IdxSkids_HR].Dosing_Pump_202.P202_GAIN := IDEC_REAL_Conv(gModbus_HR[IdxSkids_HR].Modbus_Dosing.Block8_Real[34]);
	gSkid_HR[IdxSkids_HR].Dosing_Pump_202.P202_STEPADJ := IDEC_REAL_Conv(gModbus_HR[IdxSkids_HR].Modbus_Dosing.Block8_Real[35]);
	gSkid_HR[IdxSkids_HR].Dosing_Pump_202.P202_TOTALADJ := IDEC_REAL_Conv(gModbus_HR[IdxSkids_HR].Modbus_Dosing.Block8_Real[36]);

	gSkid_HR[IdxSkids_HR].Dosing_Pump_203.P203_REF_SENSOR := IDEC_REAL_Conv(gModbus_HR[IdxSkids_HR].Modbus_Dosing.Block8_Real[38]);
	gSkid_HR[IdxSkids_HR].Dosing_Pump_203.P203_CONC := IDEC_REAL_Conv(gModbus_HR[IdxSkids_HR].Modbus_Dosing.Block8_Real[39]);
	gSkid_HR[IdxSkids_HR].Dosing_Pump_203.P203_PPM := IDEC_REAL_Conv(gModbus_HR[IdxSkids_HR].Modbus_Dosing.Block8_Real[40]);
	gSkid_HR[IdxSkids_HR].Dosing_Pump_203.P203_APPM := IDEC_REAL_Conv(gModbus_HR[IdxSkids_HR].Modbus_Dosing.Block8_Real[41]);
	gSkid_HR[IdxSkids_HR].Dosing_Pump_203.P203_SP := IDEC_REAL_Conv(gModbus_HR[IdxSkids_HR].Modbus_Dosing.Block8_Real[42]);
	gSkid_HR[IdxSkids_HR].Dosing_Pump_203.P203_PV := IDEC_REAL_Conv(gModbus_HR[IdxSkids_HR].Modbus_Dosing.Block8_Real[43]);
	gSkid_HR[IdxSkids_HR].Dosing_Pump_203.P203_OP := IDEC_REAL_Conv(gModbus_HR[IdxSkids_HR].Modbus_Dosing.Block8_Real[44]);
	gSkid_HR[IdxSkids_HR].Dosing_Pump_203.P203_PFI := IDEC_REAL_Conv(gModbus_HR[IdxSkids_HR].Modbus_Dosing.Block8_Real[45]);
	gSkid_HR[IdxSkids_HR].Dosing_Pump_203.P203_FQ := IDEC_REAL_Conv(gModbus_HR[IdxSkids_HR].Modbus_Dosing.Block8_Real[46]);
	gSkid_HR[IdxSkids_HR].Dosing_Pump_203.P203_PI := IDEC_REAL_Conv(gModbus_HR[IdxSkids_HR].Modbus_Dosing.Block8_Real[47]);
	gSkid_HR[IdxSkids_HR].Dosing_Pump_203.P203_TI := IDEC_REAL_Conv(gModbus_HR[IdxSkids_HR].Modbus_Dosing.Block8_Real[48]);
	gSkid_HR[IdxSkids_HR].Dosing_Pump_203.P203_PFQ := IDEC_REAL_Conv(gModbus_HR[IdxSkids_HR].Modbus_Dosing.Block8_Real[49]);
	gSkid_HR[IdxSkids_HR].Dosing_Pump_203.P203_PPI := IDEC_REAL_Conv(gModbus_HR[IdxSkids_HR].Modbus_Dosing.Block8_Real[50]);
	gSkid_HR[IdxSkids_HR].Dosing_Pump_203.P203_LS := IDEC_REAL_Conv(gModbus_HR[IdxSkids_HR].Modbus_Dosing.Block8_Real[51]);
	gSkid_HR[IdxSkids_HR].Dosing_Pump_203.P203_ASP := IDEC_REAL_Conv(gModbus_HR[IdxSkids_HR].Modbus_Dosing.Block8_Real[52]);
	gSkid_HR[IdxSkids_HR].Dosing_Pump_203.P203_GAIN := IDEC_REAL_Conv(gModbus_HR[IdxSkids_HR].Modbus_Dosing.Block8_Real[53]);
	gSkid_HR[IdxSkids_HR].Dosing_Pump_203.P203_STEPADJ := IDEC_REAL_Conv(gModbus_HR[IdxSkids_HR].Modbus_Dosing.Block8_Real[54]);
	gSkid_HR[IdxSkids_HR].Dosing_Pump_203.P203_TOTALADJ := IDEC_REAL_Conv(gModbus_HR[IdxSkids_HR].Modbus_Dosing.Block8_Real[55]);

	gSkid_HR[IdxSkids_HR].Dosing_Pump_204.P204_REF_SENSOR := IDEC_REAL_Conv(gModbus_HR[IdxSkids_HR].Modbus_Dosing.Block8_Real[57]);
	gSkid_HR[IdxSkids_HR].Dosing_Pump_204.P204_CONC := IDEC_REAL_Conv(gModbus_HR[IdxSkids_HR].Modbus_Dosing.Block8_Real[58]);
	gSkid_HR[IdxSkids_HR].Dosing_Pump_204.P204_PPM := IDEC_REAL_Conv(gModbus_HR[IdxSkids_HR].Modbus_Dosing.Block8_Real[59]);
	gSkid_HR[IdxSkids_HR].Dosing_Pump_204.P204_APPM := IDEC_REAL_Conv(gModbus_HR[IdxSkids_HR].Modbus_Dosing.Block8_Real[60]);
	gSkid_HR[IdxSkids_HR].Dosing_Pump_204.P204_SP := IDEC_REAL_Conv(gModbus_HR[IdxSkids_HR].Modbus_Dosing.Block8_Real[61]);
	gSkid_HR[IdxSkids_HR].Dosing_Pump_204.P204_PV := IDEC_REAL_Conv(gModbus_HR[IdxSkids_HR].Modbus_Dosing.Block8_Real[62]);

	// AS Block 9 - 7000 DOSING REAL
	gSkid_HR[IdxSkids_HR].Dosing_Pump_204.P204_OP := IDEC_REAL_Conv(gModbus_HR[IdxSkids_HR].Modbus_Dosing.Block9_Real[0]);
	gSkid_HR[IdxSkids_HR].Dosing_Pump_204.P204_PFI := IDEC_REAL_Conv(gModbus_HR[IdxSkids_HR].Modbus_Dosing.Block9_Real[1]);
	gSkid_HR[IdxSkids_HR].Dosing_Pump_204.P204_FQ := IDEC_REAL_Conv(gModbus_HR[IdxSkids_HR].Modbus_Dosing.Block9_Real[2]);
	gSkid_HR[IdxSkids_HR].Dosing_Pump_204.P204_PI := IDEC_REAL_Conv(gModbus_HR[IdxSkids_HR].Modbus_Dosing.Block9_Real[3]);
	gSkid_HR[IdxSkids_HR].Dosing_Pump_204.P204_TI := IDEC_REAL_Conv(gModbus_HR[IdxSkids_HR].Modbus_Dosing.Block9_Real[4]);
	gSkid_HR[IdxSkids_HR].Dosing_Pump_204.P204_PFQ := IDEC_REAL_Conv(gModbus_HR[IdxSkids_HR].Modbus_Dosing.Block9_Real[5]);
	gSkid_HR[IdxSkids_HR].Dosing_Pump_204.P204_PPI := IDEC_REAL_Conv(gModbus_HR[IdxSkids_HR].Modbus_Dosing.Block9_Real[6]);
	gSkid_HR[IdxSkids_HR].Dosing_Pump_204.P204_LS := IDEC_REAL_Conv(gModbus_HR[IdxSkids_HR].Modbus_Dosing.Block9_Real[7]);
	gSkid_HR[IdxSkids_HR].Dosing_Pump_204.P204_ASP := IDEC_REAL_Conv(gModbus_HR[IdxSkids_HR].Modbus_Dosing.Block9_Real[8]);
	gSkid_HR[IdxSkids_HR].Dosing_Pump_204.P204_GAIN := IDEC_REAL_Conv(gModbus_HR[IdxSkids_HR].Modbus_Dosing.Block8_Real[9]);
	gSkid_HR[IdxSkids_HR].Dosing_Pump_204.P204_STEPADJ := IDEC_REAL_Conv(gModbus_HR[IdxSkids_HR].Modbus_Dosing.Block8_Real[10]);
	gSkid_HR[IdxSkids_HR].Dosing_Pump_204.P204_TOTALADJ := IDEC_REAL_Conv(gModbus_HR[IdxSkids_HR].Modbus_Dosing.Block8_Real[11]);

	gSkid_HR[IdxSkids_HR].Dosing_Pump_205.P205_REF_SENSOR := IDEC_REAL_Conv(gModbus_HR[IdxSkids_HR].Modbus_Dosing.Block9_Real[13]);
	gSkid_HR[IdxSkids_HR].Dosing_Pump_205.P205_CONC := IDEC_REAL_Conv(gModbus_HR[IdxSkids_HR].Modbus_Dosing.Block9_Real[14]);
	gSkid_HR[IdxSkids_HR].Dosing_Pump_205.P205_PPM := IDEC_REAL_Conv(gModbus_HR[IdxSkids_HR].Modbus_Dosing.Block9_Real[15]);
	gSkid_HR[IdxSkids_HR].Dosing_Pump_205.P205_APPM := IDEC_REAL_Conv(gModbus_HR[IdxSkids_HR].Modbus_Dosing.Block9_Real[16]);
	gSkid_HR[IdxSkids_HR].Dosing_Pump_205.P205_SP := IDEC_REAL_Conv(gModbus_HR[IdxSkids_HR].Modbus_Dosing.Block9_Real[17]);
	gSkid_HR[IdxSkids_HR].Dosing_Pump_205.P205_PV := IDEC_REAL_Conv(gModbus_HR[IdxSkids_HR].Modbus_Dosing.Block9_Real[18]);
	gSkid_HR[IdxSkids_HR].Dosing_Pump_205.P205_OP := IDEC_REAL_Conv(gModbus_HR[IdxSkids_HR].Modbus_Dosing.Block9_Real[19]);
	gSkid_HR[IdxSkids_HR].Dosing_Pump_205.P205_PFI := IDEC_REAL_Conv(gModbus_HR[IdxSkids_HR].Modbus_Dosing.Block9_Real[20]);
	gSkid_HR[IdxSkids_HR].Dosing_Pump_205.P205_FQ := IDEC_REAL_Conv(gModbus_HR[IdxSkids_HR].Modbus_Dosing.Block9_Real[21]);
	gSkid_HR[IdxSkids_HR].Dosing_Pump_205.P205_PI := IDEC_REAL_Conv(gModbus_HR[IdxSkids_HR].Modbus_Dosing.Block9_Real[22]);
	gSkid_HR[IdxSkids_HR].Dosing_Pump_205.P205_TI := IDEC_REAL_Conv(gModbus_HR[IdxSkids_HR].Modbus_Dosing.Block9_Real[23]);
	gSkid_HR[IdxSkids_HR].Dosing_Pump_205.P205_PFQ := IDEC_REAL_Conv(gModbus_HR[IdxSkids_HR].Modbus_Dosing.Block9_Real[24]);
	gSkid_HR[IdxSkids_HR].Dosing_Pump_205.P205_PPI := IDEC_REAL_Conv(gModbus_HR[IdxSkids_HR].Modbus_Dosing.Block9_Real[25]);
	gSkid_HR[IdxSkids_HR].Dosing_Pump_205.P205_LS := IDEC_REAL_Conv(gModbus_HR[IdxSkids_HR].Modbus_Dosing.Block9_Real[26]);

	gSkid_HR[IdxSkids_HR].Dosing_Pump_206.P206_REF_SENSOR := IDEC_REAL_Conv(gModbus_HR[IdxSkids_HR].Modbus_Dosing.Block9_Real[32]);
	gSkid_HR[IdxSkids_HR].Dosing_Pump_206.P206_CONC := IDEC_REAL_Conv(gModbus_HR[IdxSkids_HR].Modbus_Dosing.Block9_Real[33]);
	gSkid_HR[IdxSkids_HR].Dosing_Pump_206.P206_PPM := IDEC_REAL_Conv(gModbus_HR[IdxSkids_HR].Modbus_Dosing.Block9_Real[34]);
	gSkid_HR[IdxSkids_HR].Dosing_Pump_206.P206_APPM := IDEC_REAL_Conv(gModbus_HR[IdxSkids_HR].Modbus_Dosing.Block9_Real[35]);
	gSkid_HR[IdxSkids_HR].Dosing_Pump_206.P206_SP := IDEC_REAL_Conv(gModbus_HR[IdxSkids_HR].Modbus_Dosing.Block9_Real[36]);
	gSkid_HR[IdxSkids_HR].Dosing_Pump_206.P206_PV := IDEC_REAL_Conv(gModbus_HR[IdxSkids_HR].Modbus_Dosing.Block9_Real[37]);
	gSkid_HR[IdxSkids_HR].Dosing_Pump_206.P206_OP := IDEC_REAL_Conv(gModbus_HR[IdxSkids_HR].Modbus_Dosing.Block9_Real[38]);
	gSkid_HR[IdxSkids_HR].Dosing_Pump_206.P206_PFI := IDEC_REAL_Conv(gModbus_HR[IdxSkids_HR].Modbus_Dosing.Block9_Real[39]);
	gSkid_HR[IdxSkids_HR].Dosing_Pump_206.P206_FQ := IDEC_REAL_Conv(gModbus_HR[IdxSkids_HR].Modbus_Dosing.Block9_Real[40]);
	gSkid_HR[IdxSkids_HR].Dosing_Pump_206.P206_PI := IDEC_REAL_Conv(gModbus_HR[IdxSkids_HR].Modbus_Dosing.Block9_Real[41]);
	gSkid_HR[IdxSkids_HR].Dosing_Pump_206.P206_TI := IDEC_REAL_Conv(gModbus_HR[IdxSkids_HR].Modbus_Dosing.Block9_Real[42]);
	gSkid_HR[IdxSkids_HR].Dosing_Pump_206.P206_PFQ := IDEC_REAL_Conv(gModbus_HR[IdxSkids_HR].Modbus_Dosing.Block9_Real[43]);
	gSkid_HR[IdxSkids_HR].Dosing_Pump_206.P206_PPI := IDEC_REAL_Conv(gModbus_HR[IdxSkids_HR].Modbus_Dosing.Block9_Real[44]);
	gSkid_HR[IdxSkids_HR].Dosing_Pump_206.P206_LS := IDEC_REAL_Conv(gModbus_HR[IdxSkids_HR].Modbus_Dosing.Block9_Real[45]);

	gSkid_HR[IdxSkids_HR].Dosing_Pump_207.P207_REF_SENSOR := IDEC_REAL_Conv(gModbus_HR[IdxSkids_HR].Modbus_Dosing.Block9_Real[51]);
	gSkid_HR[IdxSkids_HR].Dosing_Pump_207.P207_CONC := IDEC_REAL_Conv(gModbus_HR[IdxSkids_HR].Modbus_Dosing.Block9_Real[52]);
	gSkid_HR[IdxSkids_HR].Dosing_Pump_207.P207_PPM := IDEC_REAL_Conv(gModbus_HR[IdxSkids_HR].Modbus_Dosing.Block9_Real[53]);
	gSkid_HR[IdxSkids_HR].Dosing_Pump_207.P207_APPM := IDEC_REAL_Conv(gModbus_HR[IdxSkids_HR].Modbus_Dosing.Block9_Real[54]);
	gSkid_HR[IdxSkids_HR].Dosing_Pump_207.P207_SP := IDEC_REAL_Conv(gModbus_HR[IdxSkids_HR].Modbus_Dosing.Block9_Real[55]);
	gSkid_HR[IdxSkids_HR].Dosing_Pump_207.P207_PV := IDEC_REAL_Conv(gModbus_HR[IdxSkids_HR].Modbus_Dosing.Block9_Real[56]);
	gSkid_HR[IdxSkids_HR].Dosing_Pump_207.P207_OP := IDEC_REAL_Conv(gModbus_HR[IdxSkids_HR].Modbus_Dosing.Block9_Real[57]);
	gSkid_HR[IdxSkids_HR].Dosing_Pump_207.P207_PFI := IDEC_REAL_Conv(gModbus_HR[IdxSkids_HR].Modbus_Dosing.Block9_Real[58]);
	gSkid_HR[IdxSkids_HR].Dosing_Pump_207.P207_FQ := IDEC_REAL_Conv(gModbus_HR[IdxSkids_HR].Modbus_Dosing.Block9_Real[59]);
	gSkid_HR[IdxSkids_HR].Dosing_Pump_207.P207_PI := IDEC_REAL_Conv(gModbus_HR[IdxSkids_HR].Modbus_Dosing.Block9_Real[60]);
	gSkid_HR[IdxSkids_HR].Dosing_Pump_207.P207_TI := IDEC_REAL_Conv(gModbus_HR[IdxSkids_HR].Modbus_Dosing.Block9_Real[61]);
	gSkid_HR[IdxSkids_HR].Dosing_Pump_207.P207_PFQ := IDEC_REAL_Conv(gModbus_HR[IdxSkids_HR].Modbus_Dosing.Block9_Real[62]);

	// AS Block 10 - 7000 DOSING REAL
	gSkid_HR[IdxSkids_HR].Dosing_Pump_207.P207_PPI := IDEC_REAL_Conv(gModbus_HR[IdxSkids_HR].Modbus_Dosing.Block10_Real[0]);
	gSkid_HR[IdxSkids_HR].Dosing_Pump_207.P207_LS := IDEC_REAL_Conv(gModbus_HR[IdxSkids_HR].Modbus_Dosing.Block10_Real[1]);

	gSkid_HR[IdxSkids_HR].Dosing_Pump_208.P208_REF_SENSOR := IDEC_REAL_Conv(gModbus_HR[IdxSkids_HR].Modbus_Dosing.Block10_Real[7]);
	gSkid_HR[IdxSkids_HR].Dosing_Pump_208.P208_CONC := IDEC_REAL_Conv(gModbus_HR[IdxSkids_HR].Modbus_Dosing.Block10_Real[8]);
	gSkid_HR[IdxSkids_HR].Dosing_Pump_208.P208_PPM := IDEC_REAL_Conv(gModbus_HR[IdxSkids_HR].Modbus_Dosing.Block10_Real[9]);
	gSkid_HR[IdxSkids_HR].Dosing_Pump_208.P208_APPM := IDEC_REAL_Conv(gModbus_HR[IdxSkids_HR].Modbus_Dosing.Block10_Real[10]);
	gSkid_HR[IdxSkids_HR].Dosing_Pump_208.P208_SP := IDEC_REAL_Conv(gModbus_HR[IdxSkids_HR].Modbus_Dosing.Block10_Real[11]);
	gSkid_HR[IdxSkids_HR].Dosing_Pump_208.P208_PV := IDEC_REAL_Conv(gModbus_HR[IdxSkids_HR].Modbus_Dosing.Block10_Real[12]);
	gSkid_HR[IdxSkids_HR].Dosing_Pump_208.P208_OP := IDEC_REAL_Conv(gModbus_HR[IdxSkids_HR].Modbus_Dosing.Block10_Real[13]);
	gSkid_HR[IdxSkids_HR].Dosing_Pump_208.P208_PFI := IDEC_REAL_Conv(gModbus_HR[IdxSkids_HR].Modbus_Dosing.Block10_Real[14]);
	gSkid_HR[IdxSkids_HR].Dosing_Pump_208.P208_FQ := IDEC_REAL_Conv(gModbus_HR[IdxSkids_HR].Modbus_Dosing.Block10_Real[15]);
	gSkid_HR[IdxSkids_HR].Dosing_Pump_208.P208_PI := IDEC_REAL_Conv(gModbus_HR[IdxSkids_HR].Modbus_Dosing.Block10_Real[16]);
	gSkid_HR[IdxSkids_HR].Dosing_Pump_208.P208_TI := IDEC_REAL_Conv(gModbus_HR[IdxSkids_HR].Modbus_Dosing.Block10_Real[17]);
	gSkid_HR[IdxSkids_HR].Dosing_Pump_208.P208_PFQ := IDEC_REAL_Conv(gModbus_HR[IdxSkids_HR].Modbus_Dosing.Block10_Real[18]);
	gSkid_HR[IdxSkids_HR].Dosing_Pump_208.P208_PPI := IDEC_REAL_Conv(gModbus_HR[IdxSkids_HR].Modbus_Dosing.Block10_Real[19]);
	gSkid_HR[IdxSkids_HR].Dosing_Pump_208.P208_LS := IDEC_REAL_Conv(gModbus_HR[IdxSkids_HR].Modbus_Dosing.Block10_Real[20]);

	gSkid_HR[IdxSkids_HR].Sensor_Variables.SENSOR301 := IDEC_REAL_Conv(gModbus_HR[IdxSkids_HR].Modbus_Dosing.Block10_Real[26]);
	gSkid_HR[IdxSkids_HR].Sensor_Variables.SENSOR302 := IDEC_REAL_Conv(gModbus_HR[IdxSkids_HR].Modbus_Dosing.Block10_Real[27]);
	gSkid_HR[IdxSkids_HR].Sensor_Variables.SENSOR303 := IDEC_REAL_Conv(gModbus_HR[IdxSkids_HR].Modbus_Dosing.Block10_Real[28]);
	gSkid_HR[IdxSkids_HR].Sensor_Variables.SENSOR304 := IDEC_REAL_Conv(gModbus_HR[IdxSkids_HR].Modbus_Dosing.Block10_Real[29]);

	gSkid_HR[IdxSkids_HR].Sensor_Variables.FI301 := IDEC_REAL_Conv(gModbus_HR[IdxSkids_HR].Modbus_Dosing.Block10_Real[34]);
	gSkid_HR[IdxSkids_HR].Sensor_Variables.FI301_QT := IDEC_REAL_Conv(gModbus_HR[IdxSkids_HR].Modbus_Dosing.Block10_Real[35]);
	gSkid_HR[IdxSkids_HR].Sensor_Variables.FI302 := IDEC_REAL_Conv(gModbus_HR[IdxSkids_HR].Modbus_Dosing.Block10_Real[36]);
	gSkid_HR[IdxSkids_HR].Sensor_Variables.FI302_QT := IDEC_REAL_Conv(gModbus_HR[IdxSkids_HR].Modbus_Dosing.Block10_Real[37]);
	gSkid_HR[IdxSkids_HR].Sensor_Variables.FI303 := IDEC_REAL_Conv(gModbus_HR[IdxSkids_HR].Modbus_Dosing.Block10_Real[38]);
	gSkid_HR[IdxSkids_HR].Sensor_Variables.FI303_QT := IDEC_REAL_Conv(gModbus_HR[IdxSkids_HR].Modbus_Dosing.Block10_Real[39]);
	gSkid_HR[IdxSkids_HR].Sensor_Variables.FI304 := IDEC_REAL_Conv(gModbus_HR[IdxSkids_HR].Modbus_Dosing.Block10_Real[40]);
	gSkid_HR[IdxSkids_HR].Sensor_Variables.FI304_QT := IDEC_REAL_Conv(gModbus_HR[IdxSkids_HR].Modbus_Dosing.Block10_Real[41]);

	// AS Block 11 - 7000 DOSING REAL - SPARE
	//:= IDEC_REAL_Conv(gModbus_HR[IdxSkids_HR].Modbus_Dosing.Block11_Real[0]);

	// AS Block 48 - ALARMS
	gSkid_HR[IdxSkids_HR].Alarms.ALARM_AB1 := gModbus_HR[IdxSkids_HR].Modbus_Alarms.Block48_Int[0];
	gSkid_HR[IdxSkids_HR].Alarms.ALARM_AB2 := gModbus_HR[IdxSkids_HR].Modbus_Alarms.Block48_Int[1];
	gSkid_HR[IdxSkids_HR].Alarms.ALARM_AB3 := gModbus_HR[IdxSkids_HR].Modbus_Alarms.Block48_Int[2];
	gSkid_HR[IdxSkids_HR].Alarms.ALARM_AB4 := gModbus_HR[IdxSkids_HR].Modbus_Alarms.Block48_Int[3];
	gSkid_HR[IdxSkids_HR].Alarms.ALARM_AB5 := gModbus_HR[IdxSkids_HR].Modbus_Alarms.Block48_Int[4];
	gSkid_HR[IdxSkids_HR].Alarms.ALARM_AB6 := gModbus_HR[IdxSkids_HR].Modbus_Alarms.Block48_Int[5];
	gSkid_HR[IdxSkids_HR].Alarms.ALARM_AB7 := gModbus_HR[IdxSkids_HR].Modbus_Alarms.Block48_Int[6];
	gSkid_HR[IdxSkids_HR].Alarms.ALARM_AB8 := gModbus_HR[IdxSkids_HR].Modbus_Alarms.Block48_Int[7];
	gSkid_HR[IdxSkids_HR].Alarms.ALARM_AB9 := gModbus_HR[IdxSkids_HR].Modbus_Alarms.Block48_Int[8];
	gSkid_HR[IdxSkids_HR].Alarms.ALARM_AB10 := gModbus_HR[IdxSkids_HR].Modbus_Alarms.Block48_Int[9];
	gSkid_HR[IdxSkids_HR].Alarms.ALARM_AB11 := gModbus_HR[IdxSkids_HR].Modbus_Alarms.Block48_Int[10];

	gSkid_HR[IdxSkids_HR].Alarms.ALARM_AB12 := gModbus_HR[IdxSkids_HR].Modbus_Alarms.Block48_Int[51];
	gSkid_HR[IdxSkids_HR].Alarms.ALARM_AB13 := gModbus_HR[IdxSkids_HR].Modbus_Alarms.Block48_Int[52];
	gSkid_HR[IdxSkids_HR].Alarms.ALARM_AB14 := gModbus_HR[IdxSkids_HR].Modbus_Alarms.Block48_Int[53];
	gSkid_HR[IdxSkids_HR].Alarms.ALARM_AB15 := gModbus_HR[IdxSkids_HR].Modbus_Alarms.Block48_Int[54];
	gSkid_HR[IdxSkids_HR].Alarms.ALARM_AB16 := gModbus_HR[IdxSkids_HR].Modbus_Alarms.Block48_Int[55];
	gSkid_HR[IdxSkids_HR].Alarms.ALARM_AB17 := gModbus_HR[IdxSkids_HR].Modbus_Alarms.Block48_Int[56];
	gSkid_HR[IdxSkids_HR].Alarms.ALARM_AB18 := gModbus_HR[IdxSkids_HR].Modbus_Alarms.Block48_Int[57];
	gSkid_HR[IdxSkids_HR].Alarms.ALARM_AB19 := gModbus_HR[IdxSkids_HR].Modbus_Alarms.Block48_Int[58];

	// AS Block 61 - DOSING PUMP TEXT
	IDEC_String(ADR(gSkid_HR[IdxSkids_HR].Dosing_Pump_201.P201_TEXT),ADR(gModbus_HR[IdxSkids_HR].Modbus_Dosing.Block61_Int[0]),SIZEOF(gSkid_HR[IdxSkids_HR].Dosing_Pump_201.P201_TEXT),27);
	IDEC_String(ADR(gSkid_HR[IdxSkids_HR].Dosing_Pump_202.P202_TEXT),ADR(gModbus_HR[IdxSkids_HR].Modbus_Dosing.Block61_Int[28]),SIZEOF(gSkid_HR[IdxSkids_HR].Dosing_Pump_202.P202_TEXT),27);
	IDEC_String(ADR(gSkid_HR[IdxSkids_HR].Dosing_Pump_203.P203_TEXT),ADR(gModbus_HR[IdxSkids_HR].Modbus_Dosing.Block61_Int[56]),SIZEOF(gSkid_HR[IdxSkids_HR].Dosing_Pump_203.P203_TEXT),27);
	IDEC_String(ADR(gSkid_HR[IdxSkids_HR].Dosing_Pump_204.P204_TEXT),ADR(gModbus_HR[IdxSkids_HR].Modbus_Dosing.Block61_Int[84]),SIZEOF(gSkid_HR[IdxSkids_HR].Dosing_Pump_204.P204_TEXT),27);

END_ACTION
```

### Program Logical/modbusTCP/ModMaster (IEC)

#### ModMaster.var - Local variables
```iecst
(*-----------------------------------------------------------------------------------------------------------------------------------------------------------------------------------------------------------------------------------------*)
(*Modbus master function block and configuration*)
VAR
	ModbusTcpMaster : ARRAY[0..MAX_SKIDS] OF MBmaster;
	MasterConfig : ARRAY[0..MAX_SKIDS] OF modbus_master_cfg_typ;
	reset_error : BOOL := FALSE;
END_VAR
(*IO sample arrays*)
VAR
	A_Out : ARRAY[0..255] OF UINT := [256(0)];
	UINT_In : ARRAY[0..50] OF UINT := [51(0)];
	REAL_In : ARRAY[0..50] OF REAL := [51(0.0)];
	D_Out : ARRAY[0..255] OF BOOL := [256(FALSE)];
	D_In : ARRAY[0..255] OF BOOL := [256(FALSE)];
END_VAR
(*MISC variables*)
VAR
	interface : STRING[20];
	logger : ARRAY[0..LLN,0..MAX_SKIDS] OF STRING[LLL];
	StartStop : BOOL := FALSE;
	LREAL_Test : LREAL := 0.0;
	UDINT_Test : UDINT := 0;
	Test_REAL : ARRAY[0..3] OF REAL := [4(0)];
	Test_UDINT : UDINT := 0;
	Test_SWAPPED_UDINT : UDINT := 0;
	IdxReals : INT := 0;
	IdxUINTS : INT := 0;
	IdxSkids : INT;
	SkidString : STRING[80];
	SkidNumberINT : STRING[80];
	TestBool : BOOL;
END_VAR
```
